(* IEC 61131-3 sources: ia2/examples/sim_smoke/pous, 1 file *)

(* ---- main.st ---- *)
(* Tiny tank model: the scenario plays the plant by writing
   inlet_cmd; level integrates while it holds. Used by
   scenarios/fill.toml as the cs sim reference example. *)
PROGRAM main
  VAR
    inlet_cmd : BOOL;
    level : REAL;
    overflow : BOOL;
  END_VAR
  IF inlet_cmd THEN
    level := level + 0.5;
  END_IF;
  IF level > 80.0 THEN
    overflow := TRUE;
  END_IF;
END_PROGRAM
